FUNCTION_BLOCK Avestruz IMPLEMENTS I_AveCorredora
VAR_INPUT
    velocidad : REAL;
    tiempoCorriendo : TIME;
END_VAR
VAR
END_VAR


METHOD Correr : BOOL
Correr := TRUE;
END_METHOD

END_FUNCTION_BLOCK

(* stored: Version 1.1.0.1, ProductVersion 3.1.4024.12
   POU Avestruz: Id {a11a740d-3e87-4b3a-bb09-55f808b82ec4}, SpecialFunc None
   Method Correr: Id {e66da694-4037-4e5e-9913-2c6f351524b5} *)
